PROGRAM TEST3
VAR
END_VAR

SETUP.AXIS_FOXTROTT();

END_PROGRAM

(* stored: Version 1.1.0.1, ProductVersion 3.1.4026.18
   POU TEST3: Id {5e80ff28-a5a1-4844-b680-4a1e89a48fd6}, SpecialFunc None *)
